{attribute 'qualified_only'}
{attribute 'strict'}
{attribute 'to_string'}
TYPE E_Command :
(
	CMD_NONE := 0,
    CMD_TO_IDLE,
    CMD_TO_HV_ACTIVE,
    CMD_TO_DEMO,
    CMD_TO_LEVITATION,
    CMD_TO_MOVEMENT,
    CMD_TO_MAINTENANCE,
    CMD_EMERGENCY
);
END_TYPE

(* stored: Version 1.1.0.1
   DUT E_Command: Id {3de4f68e-3ae1-41c8-aa15-e60118ed1dc9} *)
